# EPICS autosave request: ADAndor/andorApp/Db/andorCCD_settings.req
$(P)$(R)AndorCooler
$(P)$(R)AndorAccumulatePeriod
$(P)$(R)AndorShutterMode
$(P)$(R)AndorShutterExTTL
$(P)$(R)PALFilePath
$(P)$(R)AndorPreAmpGain
$(P)$(R)AndorADCSpeed
